// TIA Portal project "DataBlocks" (V14)

(* hardware
DEVICE "S7-1200 station_1"  S7-1200 Station
   slot 0: "Rack_0"  S7-1200 Rack  Rack  V1.0
   slot 1: "PLC_1"  CPU 1214C DC/DC/DC  6ES7 214-1AG40-0XB0  V4.2
*)

// ===== PLC "PLC_1"  CPU 1214C DC/DC/DC =====

VAR_GLOBAL   // PLC tag table "Default tag table"
   "Tag_1" AT %M300.3 : Bool;
END_VAR

DATA_BLOCK "Global_DataBlock"   // DB1
{ S7_Optimized_Access := 'TRUE' }
VERSION : 0.1
   VAR
      PontoFlutuante : Real := 10.0;
      texto : String := 'Pablo';
   END_VAR
BEGIN
END_DATA_BLOCK

DATA_BLOCK "DadosInternos_DB"   // DB2
{ S7_Optimized_Access := 'TRUE' }
VERSION : 0.1
// stored: InstanceOfName DadosInternos
"DadosInternos"
BEGIN
END_DATA_BLOCK

DATA_BLOCK "DadosInternos_DB_2"   // DB3
{ S7_Optimized_Access := 'TRUE' }
VERSION : 0.1
// stored: InstanceOfName DadosInternos
"DadosInternos"
BEGIN
END_DATA_BLOCK

FUNCTION_BLOCK "DadosInternos"   // FB1, LAD
{ S7_Optimized_Access := 'TRUE' }
VERSION : 0.1
   VAR
      Resultado : Real;
   END_VAR
   VAR CONSTANT
      PI : Real := 3.14;
   END_VAR
BEGIN

REGION Network 1
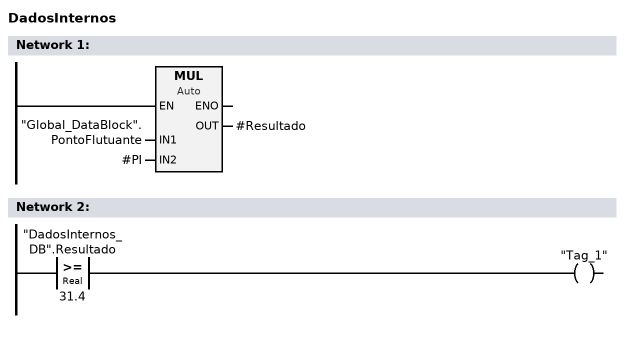
   RUNG wire#powerrail
      Mul(in1 := "Global_DataBlock".PontoFlutuante, in2 := #PI, out => #Resultado)
   END_RUNG
   // the same network as SCL:
   #Resultado := "Global_DataBlock".PontoFlutuante * #PI;
END_REGION

REGION Network 2
   RUNG wire#powerrail
      { S7_Templates := "SrcType := Real" } GE_Contact(in1 := "DadosInternos_DB".Resultado, in2 := 31.4)
      Coil( "Tag_1" )
   END_RUNG
   // the same network as SCL:
   "Tag_1" := "DadosInternos_DB".Resultado >= 31.4;
END_REGION
END_FUNCTION_BLOCK

FUNCTION "LerTexto" : Void   // FC1, LAD
{ S7_Optimized_Access := 'TRUE' }
VERSION : 0.1
   VAR_OUTPUT
      TEXTO : String;
   END_VAR
BEGIN

REGION Network 1
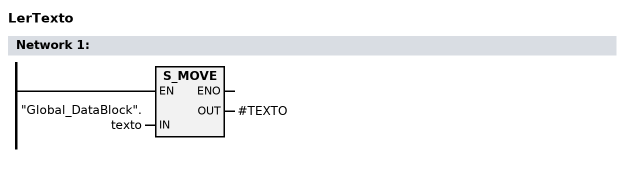
   S_MOVE(in := "Global_DataBlock".texto, out => #TEXTO);
END_REGION
END_FUNCTION

ORGANIZATION_BLOCK "Main"   // OB1, LAD, ProgramCycle
TITLE = "Main Program Sweep (Cycle)"
{ S7_Optimized_Access := 'TRUE' }
VERSION : 0.1
   VAR_INPUT
      Initial_Call : Bool;   // Initial call of this OB
      Remanence : Bool;   // =True, if remanent data are available
   END_VAR
   VAR_TEMP
      Texto : String;
   END_VAR
BEGIN

REGION Network 1
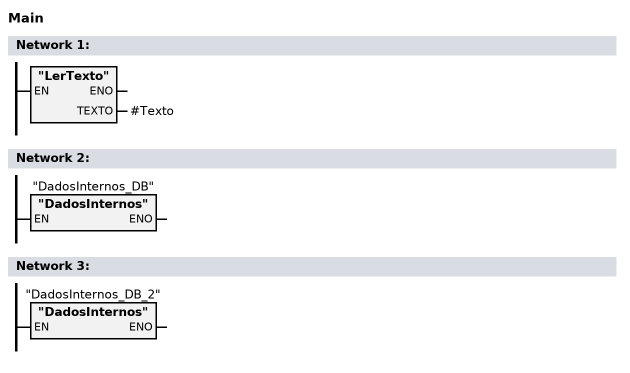
   RUNG wire#powerrail
      "LerTexto"(TEXTO => #Texto)
   END_RUNG
   // the same network as SCL:
   "LerTexto"(TEXTO => #Texto);
END_REGION

REGION Network 2
   RUNG wire#powerrail
      "DadosInternos_DB"()
   END_RUNG
   // the same network as SCL:
   "DadosInternos_DB"();   // "DadosInternos"
END_REGION

REGION Network 3
   RUNG wire#powerrail
      "DadosInternos_DB_2"()
   END_RUNG
   // the same network as SCL:
   "DadosInternos_DB_2"();   // "DadosInternos"
END_REGION
END_ORGANIZATION_BLOCK